
// ===== library: MasterCopy "fc_gw_alive_system" =====

// folder: gw_alive_system

FUNCTION "fc_gw_alive_system" : Void   // FC20, FBD
{ S7_Optimized_Access := 'TRUE' }
VERSION : 0.6
   VAR_INPUT
      alive_rcv : Bool;
      quitt_erforderlich : Bool;
      reset : Bool;
      rcv_time : Time;
      send_time : Time;
      initial_call : Bool;
   END_VAR
   VAR_OUTPUT
      alive_ok : Bool;
   END_VAR
   VAR_IN_OUT
      alive_send : Bool;
      IDB_timer : "udt_gw_alive_timer";
   END_VAR
   VAR_TEMP
      Ton_Dn : Bool;
      Toff_Dn : Bool;
      quitt : Bool;
      alive_falling : Bool;
      tcon_done_edge : Bool;
      tcon_error_edge : Bool;
      tdis_done_edge : Bool;
      tdis_error_edge : Bool;
      window_in : Bool;
      pause_in : Bool;
      pause_pt : Time;
      tcon_done : Bool;
      tcon_busy : Bool;
      tcon_error : Bool;
      tdis_done : Bool;
      tdis_busy : Bool;
      tdis_error : Bool;
      i : Int;
      tus_done : Bool;
      tus_busy : Bool;
      tus_error : Bool;
      tus_status : Word;
      tur_ndr : Bool;
      tur_busy : Bool;
      tur_error : Bool;
      tur_status : Word;
      tur_len : UDInt;
      ntp_sec : UDInt;
      unix_sec : UDInt;
      frac : UDInt;
      ns : LInt;
      lt : LTime;
      ldt_base : LDT;
      ldt_out : LDT;
      wr_ret : Int;
      b0 : UDInt;
      b1 : UDInt;
      b2 : UDInt;
      b3 : UDInt;
   END_VAR
BEGIN

REGION Network 1
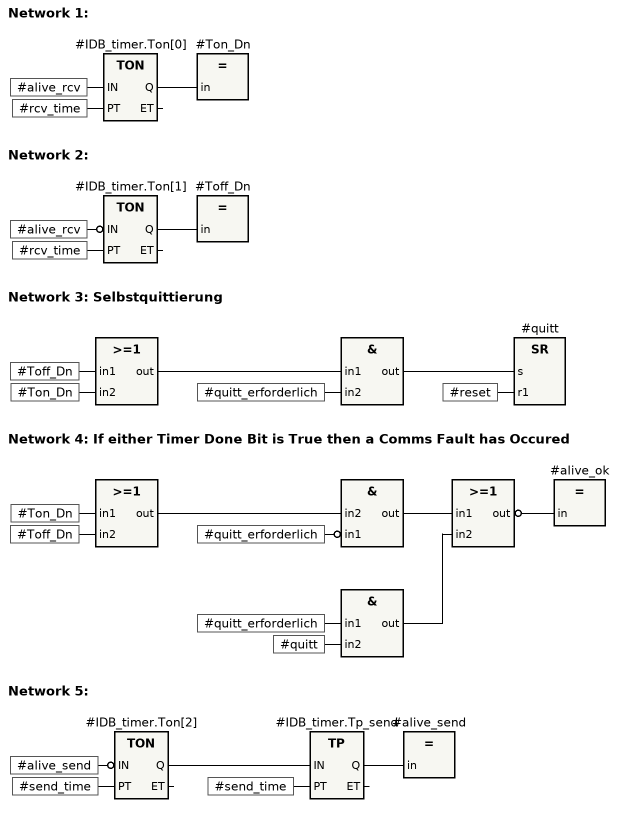
   #IDB_timer.Ton[0].TON(IN := #alive_rcv, PT := #rcv_time);
   #Ton_Dn := #IDB_timer.Ton[0].Q;
END_REGION

REGION Network 2
   #IDB_timer.Ton[1].TON(IN := NOT #alive_rcv, PT := #rcv_time);
   #Toff_Dn := #IDB_timer.Ton[1].Q;
END_REGION

REGION Network 3: Selbstquittierung
   IF (#Toff_Dn OR #Ton_Dn) AND #quitt_erforderlich THEN
       #quitt := TRUE;   // SR flip-flop
   END_IF;
   IF #reset THEN #quitt := FALSE; END_IF;
END_REGION

REGION Network 4: If either Timer Done Bit is True then a Comms Fault has Occured
   #alive_ok := NOT (((#Ton_Dn OR #Toff_Dn) AND NOT #quitt_erforderlich) OR (#quitt_erforderlich AND #quitt));
END_REGION

REGION Network 5
   #IDB_timer.Ton[2].TON(IN := NOT #alive_send, PT := #send_time);
   #IDB_timer.Tp_send.TP(IN := #IDB_timer.Ton[2].Q, PT := #send_time);
   #alive_send := #IDB_timer.Tp_send.Q;
END_REGION

REGION Network 6 (SCL): NTP sync (UDP)

   //------------------------created by cursor / 2026-08-03------------------------

   #alive_falling := "db_gw_alive_system".udp_ntp.alive_ok_prev AND NOT #alive_ok;
   #tcon_done_edge := "TCON_DB".DONE AND NOT "db_gw_alive_system".udp_ntp.tcon_done_prev;
   #tcon_error_edge := "TCON_DB".ERROR AND NOT "db_gw_alive_system".udp_ntp.tcon_error_prev;
   "db_gw_alive_system".udp_ntp.tcon_done_prev := "TCON_DB".DONE;
   "db_gw_alive_system".udp_ntp.tcon_error_prev := "TCON_DB".ERROR;
   #tdis_done_edge := "TDISCON_DB".DONE AND NOT "db_gw_alive_system".udp_ntp.tdis_done_prev;
   #tdis_error_edge := "TDISCON_DB".ERROR AND NOT "db_gw_alive_system".udp_ntp.tdis_error_prev;
   "db_gw_alive_system".udp_ntp.tdis_done_prev := "TDISCON_DB".DONE;
   "db_gw_alive_system".udp_ntp.tdis_error_prev := "TDISCON_DB".ERROR;
   IF #alive_falling AND ("db_gw_alive_system".udp_ntp.phase = 2) THEN
       "db_gw_alive_system".udp_ntp.phase := 1;
       "db_gw_alive_system".udp_ntp_cfg.conn_id := "db_gw_alive_system".udp_ntp_cfg.tcon_param.ID;
       FOR #i := 1 TO 4 DO
           "db_gw_alive_system".udp_ntp_cfg.remote_addr.REM_IP_ADDR[#i] := "db_gw_alive_system".udp_ntp_cfg.tcon_param.RemoteAddress.ADDR[#i];
       END_FOR;
       "db_gw_alive_system".udp_ntp_cfg.remote_addr.REM_PORT_NR := "db_gw_alive_system".udp_ntp_cfg.tcon_param.RemotePort;
       "db_gw_alive_system".udp_ntp.sync_done_this_window := FALSE;
       "db_gw_alive_system".udp_ntp.query_state := 0;
       "db_gw_alive_system".udp_ntp.connected := FALSE;
       "db_gw_alive_system".udp_ntp.tcon_ok := FALSE;
       "db_gw_alive_system".udp_ntp.send_req := FALSE;
       "db_gw_alive_system".udp_ntp.receive_enable := FALSE;
       "db_gw_alive_system".udp_ntp.tcon_req := FALSE;
       "db_gw_alive_system".udp_ntp.tcon_armed := FALSE;
       "db_gw_alive_system".udp_ntp.tcon_retry_wait := FALSE;
       "db_gw_alive_system".udp_ntp.time_set_done := FALSE;
       "db_gw_alive_system".udp_ntp.tdiscon_req := TRUE;
       "db_gw_alive_system".udp_ntp.tcon_after_discon := TRUE;
   ELSIF ("db_gw_alive_system".udp_ntp.phase = 0) THEN
       "db_gw_alive_system".udp_ntp.phase := 1;
       "db_gw_alive_system".udp_ntp_cfg.conn_id := "db_gw_alive_system".udp_ntp_cfg.tcon_param.ID;
       FOR #i := 1 TO 4 DO
           "db_gw_alive_system".udp_ntp_cfg.remote_addr.REM_IP_ADDR[#i] := "db_gw_alive_system".udp_ntp_cfg.tcon_param.RemoteAddress.ADDR[#i];
       END_FOR;
       "db_gw_alive_system".udp_ntp_cfg.remote_addr.REM_PORT_NR := "db_gw_alive_system".udp_ntp_cfg.tcon_param.RemotePort;
       "db_gw_alive_system".udp_ntp.sync_done_this_window := FALSE;
       "db_gw_alive_system".udp_ntp.query_state := 0;
       "db_gw_alive_system".udp_ntp.connected := FALSE;
       "db_gw_alive_system".udp_ntp.tcon_ok := FALSE;
       "db_gw_alive_system".udp_ntp.send_req := FALSE;
       "db_gw_alive_system".udp_ntp.receive_enable := FALSE;
       "db_gw_alive_system".udp_ntp.tcon_req := FALSE;
       "db_gw_alive_system".udp_ntp.tcon_armed := FALSE;
       "db_gw_alive_system".udp_ntp.tcon_retry_wait := FALSE;
       "db_gw_alive_system".udp_ntp.time_set_done := FALSE;
       "db_gw_alive_system".udp_ntp.tdiscon_req := TRUE;
       "db_gw_alive_system".udp_ntp.tcon_after_discon := TRUE;
   END_IF;
   #window_in := ("db_gw_alive_system".udp_ntp.phase = 1);
   #pause_in := ("db_gw_alive_system".udp_ntp.phase = 2);
   #pause_pt := t#3m;
   IF #alive_ok THEN
     #pause_pt := "db_gw_alive_system".udp_ntp_cfg.period_alive;
   END_IF;
   "db_gw_alive_system".udp_ntp.ton_window(IN := #window_in,
                                        PT := t#15s);
   "db_gw_alive_system".udp_ntp.ton_pause(IN := #pause_in,
                                       PT := #pause_pt);
   IF ("db_gw_alive_system".udp_ntp.phase = 1) THEN
       "db_gw_alive_system".udp_ntp.window_active := TRUE;
       IF "db_gw_alive_system".udp_ntp.tcon_armed AND NOT "db_gw_alive_system".udp_ntp.tcon_ok AND NOT "db_gw_alive_system".udp_ntp.tdiscon_req AND NOT "db_gw_alive_system".udp_ntp.tcon_after_discon AND NOT "db_gw_alive_system".udp_ntp.tcon_retry_wait AND NOT "TCON_DB".BUSY AND NOT "TDISCON_DB".BUSY THEN
           "db_gw_alive_system".udp_ntp.tcon_req := TRUE;
           "db_gw_alive_system".udp_ntp.tcon_armed := FALSE;
       END_IF;
       IF "db_gw_alive_system".udp_ntp.tcon_retry_wait AND NOT "db_gw_alive_system".udp_ntp.tcon_ok AND NOT "db_gw_alive_system".udp_ntp.tdiscon_req AND NOT "db_gw_alive_system".udp_ntp.tcon_after_discon AND ("db_gw_alive_system".udp_ntp.ton_window.ET >= "db_gw_alive_system".udp_ntp.tcon_retry_et_target) THEN
           "db_gw_alive_system".udp_ntp.tcon_armed := TRUE;
           "db_gw_alive_system".udp_ntp.tcon_retry_wait := FALSE;
       END_IF;
   ELSIF ("db_gw_alive_system".udp_ntp.phase = 2) THEN
       "db_gw_alive_system".udp_ntp.window_active := FALSE;
       "db_gw_alive_system".udp_ntp.tcon_req := FALSE;
       "db_gw_alive_system".udp_ntp.tcon_armed := FALSE;
       "db_gw_alive_system".udp_ntp.tcon_retry_wait := FALSE;
       "db_gw_alive_system".udp_ntp.send_req := FALSE;
       "db_gw_alive_system".udp_ntp.receive_enable := FALSE;
       IF "db_gw_alive_system".udp_ntp.ton_pause.Q THEN
           "db_gw_alive_system".udp_ntp.phase := 1;
           "db_gw_alive_system".udp_ntp_cfg.conn_id := "db_gw_alive_system".udp_ntp_cfg.tcon_param.ID;
           FOR #i := 1 TO 4 DO
               "db_gw_alive_system".udp_ntp_cfg.remote_addr.REM_IP_ADDR[#i] := "db_gw_alive_system".udp_ntp_cfg.tcon_param.RemoteAddress.ADDR[#i];
           END_FOR;
           "db_gw_alive_system".udp_ntp_cfg.remote_addr.REM_PORT_NR := "db_gw_alive_system".udp_ntp_cfg.tcon_param.RemotePort;
           "db_gw_alive_system".udp_ntp.sync_done_this_window := FALSE;
           "db_gw_alive_system".udp_ntp.query_state := 0;
           "db_gw_alive_system".udp_ntp.connected := FALSE;
           "db_gw_alive_system".udp_ntp.tcon_ok := FALSE;
           "db_gw_alive_system".udp_ntp.send_req := FALSE;
           "db_gw_alive_system".udp_ntp.receive_enable := FALSE;
           "db_gw_alive_system".udp_ntp.tcon_req := FALSE;
           "db_gw_alive_system".udp_ntp.tcon_armed := FALSE;
           "db_gw_alive_system".udp_ntp.tcon_retry_wait := FALSE;
           "db_gw_alive_system".udp_ntp.time_set_done := FALSE;
           "db_gw_alive_system".udp_ntp.tdiscon_req := TRUE;
           "db_gw_alive_system".udp_ntp.tcon_after_discon := TRUE;
       END_IF;
   END_IF;
   IF #tcon_done_edge AND ("TCON_DB".STATUS = 16#0000) THEN
       "db_gw_alive_system".udp_ntp.tcon_ok := TRUE;
       "db_gw_alive_system".udp_ntp.tcon_retry_wait := FALSE;
       "db_gw_alive_system".udp_ntp.tcon_after_discon := FALSE;
   END_IF;
   IF #tcon_error_edge THEN
       "db_gw_alive_system".udp_ntp.connected := FALSE;
       "db_gw_alive_system".udp_ntp.tcon_ok := FALSE;
       "db_gw_alive_system".udp_ntp.tcon_armed := FALSE;
       "db_gw_alive_system".udp_ntp.tcon_req := FALSE;
       "db_gw_alive_system".udp_ntp.send_req := FALSE;
       "db_gw_alive_system".udp_ntp.receive_enable := FALSE;
       "db_gw_alive_system".udp_ntp.query_state := 0;
       IF "db_gw_alive_system".udp_ntp.window_active THEN
           "db_gw_alive_system".udp_ntp.tdiscon_req := TRUE;
           "db_gw_alive_system".udp_ntp.tcon_after_discon := TRUE;
           "db_gw_alive_system".udp_ntp.tcon_retry_wait := TRUE;
       END_IF;
   END_IF;
   IF #tdis_done_edge OR #tdis_error_edge THEN
       "db_gw_alive_system".udp_ntp.tdiscon_req := FALSE;
       "db_gw_alive_system".udp_ntp.connected := FALSE;
       "db_gw_alive_system".udp_ntp.tcon_ok := FALSE;
       IF "db_gw_alive_system".udp_ntp.tcon_after_discon THEN
           "db_gw_alive_system".udp_ntp.tcon_after_discon := FALSE;
           IF "db_gw_alive_system".udp_ntp.window_active THEN
               IF "db_gw_alive_system".udp_ntp.tcon_retry_wait THEN
                   "db_gw_alive_system".udp_ntp.tcon_retry_et_target := "db_gw_alive_system".udp_ntp.ton_window.ET + t#2s;
               ELSE
                   "db_gw_alive_system".udp_ntp.tcon_armed := TRUE;
               END_IF;
           END_IF;
       END_IF;
   END_IF;
   IF "db_gw_alive_system".udp_ntp.reconnect_req THEN
       "db_gw_alive_system".udp_ntp.reconnect_req := FALSE;
       "db_gw_alive_system".udp_ntp.connected := FALSE;
       "db_gw_alive_system".udp_ntp.tcon_ok := FALSE;
       "db_gw_alive_system".udp_ntp.tcon_armed := FALSE;
       "db_gw_alive_system".udp_ntp.tcon_req := FALSE;
       "db_gw_alive_system".udp_ntp.send_req := FALSE;
       "db_gw_alive_system".udp_ntp.receive_enable := FALSE;
       IF "db_gw_alive_system".udp_ntp.window_active THEN
           "db_gw_alive_system".udp_ntp.tdiscon_req := TRUE;
           "db_gw_alive_system".udp_ntp.tcon_after_discon := TRUE;
           "db_gw_alive_system".udp_ntp.tcon_retry_wait := TRUE;
           "db_gw_alive_system".udp_ntp.query_state := 0;
           "db_gw_alive_system".udp_ntp.sync_done_this_window := FALSE;
       END_IF;
   END_IF;
   "TCON_DB"(REQ := "db_gw_alive_system".udp_ntp.tcon_req,
             ID := "db_gw_alive_system".udp_ntp_cfg.conn_id,
             CONNECT := "db_gw_alive_system".udp_ntp_cfg.tcon_param,
             DONE => #tcon_done,
             BUSY => #tcon_busy,
             ERROR => #tcon_error,
             STATUS => "db_gw_alive_system".udp_ntp.last_status);
   "db_gw_alive_system".udp_ntp.tcon_req := FALSE;
   "TDISCON_DB"(REQ := "db_gw_alive_system".udp_ntp.tdiscon_req,
                ID := "db_gw_alive_system".udp_ntp_cfg.conn_id,
                DONE => #tdis_done,
                BUSY => #tdis_busy,
                ERROR => #tdis_error,
                STATUS => "db_gw_alive_system".udp_ntp.last_status);
   IF NOT "db_gw_alive_system".udp_ntp.packet_ready THEN
       "db_gw_alive_system".udp_ntp.tx_buf[0] := 27;
       FOR #i := 1 TO 47 DO
           "db_gw_alive_system".udp_ntp.tx_buf[#i] := 0;
       END_FOR;
       "db_gw_alive_system".udp_ntp.packet_ready := TRUE;
   END_IF;
   IF NOT "db_gw_alive_system".udp_ntp.window_active OR "db_gw_alive_system".udp_ntp.sync_done_this_window THEN
       "db_gw_alive_system".udp_ntp.send_req := FALSE;
       "db_gw_alive_system".udp_ntp.receive_enable := FALSE;
   ELSIF NOT "db_gw_alive_system".udp_ntp.tcon_ok THEN
       "db_gw_alive_system".udp_ntp.send_req := FALSE;
       "db_gw_alive_system".udp_ntp.receive_enable := FALSE;
       "db_gw_alive_system".udp_ntp.query_state := 0;
   ELSE
       "TURCV_DB".TURCV(EN_R := "db_gw_alive_system".udp_ntp.receive_enable,
                                ID := "db_gw_alive_system".udp_ntp_cfg.conn_id,
                                LEN := 48,
                                DATA := "db_gw_alive_system".udp_ntp.rx_buf,
                                ADDR := "db_gw_alive_system".udp_ntp_cfg.remote_addr,
                                NDR => #tur_ndr,
                                BUSY => #tur_busy,
                                ERROR => #tur_error,
                                STATUS => #tur_status,
                                RCVD_LEN => #tur_len);
   "db_gw_alive_system".udp_ntp.last_status := #tur_status;
   "TUSEND_DB".TUSEND(REQ := "db_gw_alive_system".udp_ntp.send_req,
                                      ID := "db_gw_alive_system".udp_ntp_cfg.conn_id,
                                      LEN := 48,
                                      DATA := "db_gw_alive_system".udp_ntp.tx_buf,
                                      ADDR := "db_gw_alive_system".udp_ntp_cfg.remote_addr,
                                      DONE => #tus_done,
                                      BUSY => #tus_busy,
                                      ERROR => #tus_error,
                                      STATUS => #tus_status);
   "db_gw_alive_system".udp_ntp.last_status := #tus_status;
   IF (#tus_busy OR #tus_done OR #tus_error) THEN
   "db_gw_alive_system".udp_ntp.send_req := FALSE;
   END_IF;
   CASE "db_gw_alive_system".udp_ntp.query_state OF
           0:
               "db_gw_alive_system".udp_ntp.receive_enable := TRUE;
               "db_gw_alive_system".udp_ntp.rx_arm_cnt := 0;
               "db_gw_alive_system".udp_ntp.query_state := 1;
           1:
                           "db_gw_alive_system".udp_ntp.last_status := #tur_status;
               "db_gw_alive_system".udp_ntp.rx_arm_cnt := "db_gw_alive_system".udp_ntp.rx_arm_cnt + 1;
               IF "db_gw_alive_system".udp_ntp.rx_arm_cnt >= 8 THEN
                   "db_gw_alive_system".udp_ntp.send_req := TRUE;
                   "db_gw_alive_system".udp_ntp.query_state := 2;
               END_IF;
           2:
                           "db_gw_alive_system".udp_ntp.last_status := #tur_status;
               IF #tur_ndr THEN
                   "db_gw_alive_system".udp_ntp.connected := TRUE;
                   "db_gw_alive_system".udp_ntp.last_rcvd_len := #tur_len;
                   "db_gw_alive_system".udp_ntp.receive_enable := FALSE;
                   IF #tur_len = 48 THEN
                       "db_gw_alive_system".udp_ntp.query_state := 3;
                   ELSE
                       "db_gw_alive_system".udp_ntp.query_state := 0;
                   END_IF;
               ELSIF #tur_error THEN
                   "db_gw_alive_system".udp_ntp.fail_cnt := "db_gw_alive_system".udp_ntp.fail_cnt + 1;
                   IF "db_gw_alive_system".udp_ntp.fail_cnt >= 3 THEN
                       "db_gw_alive_system".udp_ntp.reconnect_req := TRUE;
                       "db_gw_alive_system".udp_ntp.fail_cnt := 0;
                   END_IF;
                   "db_gw_alive_system".udp_ntp.query_state := 0;
               ELSE
                                   "db_gw_alive_system".udp_ntp.last_status := #tus_status;
                   IF #tus_busy OR #tus_done OR #tus_error THEN
                       "db_gw_alive_system".udp_ntp.send_req := FALSE;
                   END_IF;
                   IF #tus_done THEN
                       "db_gw_alive_system".udp_ntp.receive_enable := TRUE;
                       "db_gw_alive_system".udp_ntp.rx_wait_deadline := "db_gw_alive_system".udp_ntp.ton_window.ET + t#2s;
                       "db_gw_alive_system".udp_ntp.query_state := 4;
                   ELSIF #tus_error THEN
                       "db_gw_alive_system".udp_ntp.fail_cnt := "db_gw_alive_system".udp_ntp.fail_cnt + 1;
                       IF "db_gw_alive_system".udp_ntp.fail_cnt >= 3 THEN
                           "db_gw_alive_system".udp_ntp.reconnect_req := TRUE;
                           "db_gw_alive_system".udp_ntp.fail_cnt := 0;
                       END_IF;
                       "db_gw_alive_system".udp_ntp.query_state := 0;
                   ELSIF NOT #tus_busy AND NOT #tus_done AND #tus_status = 16#7000 THEN
                       "db_gw_alive_system".udp_ntp.send_req := FALSE;
                       "db_gw_alive_system".udp_ntp.query_state := 0;
                   END_IF;
               END_IF;
           4:
                           "db_gw_alive_system".udp_ntp.last_status := #tur_status;
               IF #tur_ndr THEN
                   "db_gw_alive_system".udp_ntp.connected := TRUE;
                   "db_gw_alive_system".udp_ntp.last_rcvd_len := #tur_len;
                   "db_gw_alive_system".udp_ntp.receive_enable := FALSE;
                   "db_gw_alive_system".udp_ntp.rx_wait_deadline := t#0ms;
                   IF #tur_len = 48 THEN
                       "db_gw_alive_system".udp_ntp.query_state := 3;
                   ELSE
                       "db_gw_alive_system".udp_ntp.query_state := 0;
                   END_IF;
               ELSIF #tur_error THEN
                   "db_gw_alive_system".udp_ntp.receive_enable := FALSE;
                   "db_gw_alive_system".udp_ntp.fail_cnt := "db_gw_alive_system".udp_ntp.fail_cnt + 1;
                   IF "db_gw_alive_system".udp_ntp.fail_cnt >= 3 THEN
                       "db_gw_alive_system".udp_ntp.reconnect_req := TRUE;
                       "db_gw_alive_system".udp_ntp.fail_cnt := 0;
                   END_IF;
                   "db_gw_alive_system".udp_ntp.query_state := 0;
               ELSIF ("db_gw_alive_system".udp_ntp.rx_wait_deadline <> t#0ms) AND ("db_gw_alive_system".udp_ntp.ton_window.ET >= "db_gw_alive_system".udp_ntp.rx_wait_deadline) THEN
                   "db_gw_alive_system".udp_ntp.query_state := 0;
                   "db_gw_alive_system".udp_ntp.rx_wait_deadline := t#0ms;
               END_IF;
       END_CASE;
       IF "db_gw_alive_system".udp_ntp.query_state = 3 THEN
           #b0 := "db_gw_alive_system".udp_ntp.rx_buf[40];
           #b1 := "db_gw_alive_system".udp_ntp.rx_buf[41];
           #b2 := "db_gw_alive_system".udp_ntp.rx_buf[42];
           #b3 := "db_gw_alive_system".udp_ntp.rx_buf[43];
           #ntp_sec := #b0 * 256 + #b1;
           #ntp_sec := #ntp_sec * 256 + #b2;
           #ntp_sec := #ntp_sec * 256 + #b3;
           #b0 := "db_gw_alive_system".udp_ntp.rx_buf[44];
           #b1 := "db_gw_alive_system".udp_ntp.rx_buf[45];
           #b2 := "db_gw_alive_system".udp_ntp.rx_buf[46];
           #b3 := "db_gw_alive_system".udp_ntp.rx_buf[47];
           #frac := #b0 * 256 + #b1;
           #frac := #frac * 256 + #b2;
           #frac := #frac * 256 + #b3;
           IF #ntp_sec >= 2208988800 THEN
               #unix_sec := #ntp_sec - 2208988800;
           ELSE
               #unix_sec := #ntp_sec + 2085978496;
           END_IF;
           #ns := (LINT#1000000000 * #frac) / LINT#4294967296;
           #lt := LTIME#1s * #unix_sec + LTIME#1ns * #ns;
           #ldt_base := LDT#1970-01-01-0:0:0.0;
           #ldt_out := #ldt_base + #lt;
           "db_gw_alive_system".udp_ntp.received_time := #ldt_out;
           "db_gw_alive_system".udp_ntp.received_time_valid := TRUE;
           #wr_ret := WR_SYS_T(IN := #ldt_out);
           IF #wr_ret = 0 THEN
               IF "db_gw_alive_system".udp_ntp.sync_count < 4294967295 THEN
                   "db_gw_alive_system".udp_ntp.sync_count := "db_gw_alive_system".udp_ntp.sync_count + 1;
               END_IF;
               "db_gw_alive_system".udp_ntp.time_set_done := TRUE;
               "db_gw_alive_system".udp_ntp.sync_done_this_window := TRUE;
               "db_gw_alive_system".udp_ntp.fail_cnt := 0;
               "db_gw_alive_system".udp_ntp.query_state := 0;
           ELSE
               "db_gw_alive_system".udp_ntp.last_status := INT_TO_WORD(IN := #wr_ret);
               "db_gw_alive_system".udp_ntp.query_state := 0;
           END_IF;
       END_IF;
   END_IF;
   IF ("db_gw_alive_system".udp_ntp.phase = 1) AND ("db_gw_alive_system".udp_ntp.ton_window.Q OR "db_gw_alive_system".udp_ntp.time_set_done) THEN
       "db_gw_alive_system".udp_ntp.tcon_req := FALSE;
       "db_gw_alive_system".udp_ntp.tcon_armed := FALSE;
       "db_gw_alive_system".udp_ntp.tcon_retry_wait := FALSE;
       "db_gw_alive_system".udp_ntp.tcon_after_discon := FALSE;
       "db_gw_alive_system".udp_ntp.send_req := FALSE;
       "db_gw_alive_system".udp_ntp.receive_enable := FALSE;
       "db_gw_alive_system".udp_ntp.query_state := 0;
       "db_gw_alive_system".udp_ntp.tdiscon_req := TRUE;
       "db_gw_alive_system".udp_ntp.window_active := FALSE;
       "db_gw_alive_system".udp_ntp.tcon_ok := FALSE;
       "db_gw_alive_system".udp_ntp.time_set_done := FALSE;
       "db_gw_alive_system".udp_ntp.phase := 2;
   END_IF;
   "db_gw_alive_system".udp_ntp.alive_ok_prev := #alive_ok;
END_REGION
END_FUNCTION

// ===== library: MasterCopy "db_gw_alive_system" =====

// folder: gw_alive_system

DATA_BLOCK "db_gw_alive_system"   // DB2
{ S7_Optimized_Access := 'TRUE' }
VERSION : 0.5
   VAR
      "timer" : "udt_gw_alive_timer";
   END_VAR
   VAR RETAIN
      udp_ntp_cfg : Struct   // Retain NTP connection config — edit tcon_param only; conn_id/remote_addr synced in FC
         tcon_param : TCON_IP_v4;   // Retain source of truth: InterfaceId, ID, IP, ports (edit only here)
         conn_id : CONN_OUC := 1;   // Synced from tcon_param.ID at NTP window start
         remote_addr : TADDR_Param;   // Synced from tcon_param RemoteAddress/RemotePort at NTP window start
         period_alive : Time := T#3H;   // NTP Pause if alive_ok=TRUE
      END_STRUCT;
   END_VAR
   VAR
      udp_ntp : Struct
         alive_ok_prev : Bool;   // Previous-cycle alive_ok for falling-edge detection
         phase : Int := 0;   // 0=Idle, 1=NTP window 15s, 2=pause (!alive:T#3m / alive:period_alive)
         ton_window : TON_TIME;   // Active NTP window timer (TON, PT=T#15s)
         ton_pause : TON_TIME;   // Pause: T#3m if !alive_ok; period_alive if alive_ok
         window_active : Bool;   // TRUE while phase=1 (NTP query allowed)
         connected : Bool;   // TRUE only after NTP reply (TURCV NDR) — not after TCON alone
         tcon_ok : Bool;   // TRUE after TCON DONE+STATUS0 (UDP endpoint); allows send/receive
         tcon_armed : Bool;   // One-shot: next cycle may pulse tcon_req
         tcon_retry_wait : Bool;   // Waiting for retry cooldown after TCON/query failure
         tcon_retry_et_target : Time;   // ton_window.ET value when TCON may be re-armed
         tcon_after_discon : Bool;   // After TDISCON completes, continue with TCON/retry
         tcon_req : Bool;   // TCON REQ pulse (rising edge)
         tcon_done_prev : Bool;   // Edge memory for TCON DONE
         tcon_error_prev : Bool;   // Edge memory for TCON ERROR
         tdiscon_req : Bool;   // TDISCON REQ (held until DONE/ERROR)
         tdis_done_prev : Bool;   // Edge memory for TDISCON DONE
         tdis_error_prev : Bool;   // Edge memory for TDISCON ERROR
         reconnect_req : Bool;   // Set on TUSEND/TURCV failure (inline reconnect)
         packet_ready : Bool;   // NTP request buffer initialized once
         send_req : Bool;   // TUSEND REQ
         receive_enable : Bool;   // TURCV EN_R
         query_state : Int;   // 0=start send, 1=TUSEND, 2=TURCV, 3=parse/set time
         rx_wait_deadline : Time;   // ton_window.ET deadline to resend if no TURCV NDR
         sync_done_this_window : Bool;   // NTP sync finished for current window
         time_set_done : Bool;   // WR_SYS_T succeeded in current window
         received_time : LDT;   // Last parsed NTP transmit timestamp
         received_time_valid : Bool;   // received_time is valid
         sync_count : UDInt;   // Successful WR_SYS_T count (saturates, no wrap)
         last_rcvd_len : UDInt;   // Last TURCV RCVD_LEN (diag)
         rx_arm_cnt : Int;   // TURCV arm cycles before first TUSEND
         fail_cnt : Int;   // Consecutive fails before reconnect
         last_status : Word;   // Last TUSEND/TURCV/WR_SYS_T status
         tx_buf : Array[0..47] of Byte;   // NTP client request (48 bytes)
         rx_buf : Array[0..47] of Byte;   // NTP server response (48 bytes)
      END_STRUCT;
   END_VAR
BEGIN
   udp_ntp_cfg.tcon_param.InterfaceId := 64;
   udp_ntp_cfg.tcon_param.ID := 1;
   udp_ntp_cfg.tcon_param.ConnectionType := 19;
   udp_ntp_cfg.tcon_param.ActiveEstablished := false;
   udp_ntp_cfg.tcon_param.RemoteAddress.ADDR[1] := 10;
   udp_ntp_cfg.tcon_param.RemoteAddress.ADDR[2] := 11;
   udp_ntp_cfg.tcon_param.RemoteAddress.ADDR[3] := 2;
   udp_ntp_cfg.tcon_param.RemoteAddress.ADDR[4] := 1;
   udp_ntp_cfg.tcon_param.RemotePort := 123;
   udp_ntp_cfg.tcon_param.LocalPort := 2000;
   udp_ntp_cfg.remote_addr.REM_IP_ADDR[1] := 10;
   udp_ntp_cfg.remote_addr.REM_IP_ADDR[2] := 11;
   udp_ntp_cfg.remote_addr.REM_IP_ADDR[3] := 2;
   udp_ntp_cfg.remote_addr.REM_IP_ADDR[4] := 1;
   udp_ntp_cfg.remote_addr.REM_PORT_NR := 123;
   udp_ntp.tx_buf[0] := 16#1B;
END_DATA_BLOCK

// ===== library: MasterCopy "udt_gw_alive_timer" =====

TYPE "udt_gw_alive_timer"
   STRUCT
      Ton : Array[0..2] of TON_TIME;
      Tp_send : TP_TIME;
   END_STRUCT;
END_TYPE